(* CoDeSys 2.3.9.48 project: 5_hospital-Vyt_1Item.pro *)
(* Libraries: Standard.lib 8.11.10 13:37:48 *)

(* PLC configuration (modules and I/O channels)
_Y1_1 AT %QX0.0 [BOOLOnX_Q] Ch_1 Digital output
_Y2_1 AT %QX0.1 [BOOLOnX_Q] Ch_2 Digital output
_PCH1_1 AT %QX0.2 [BOOLOnX_Q] Ch_3 Digital output
_PCH2_1 AT %QX0.3 [BOOLOnX_Q] Ch_4 Digital output
AT %QX0.4 [BOOLOnX_Q] Ch_5 Digital output
AT %QX0.5 [BOOLOnX_Q] Ch_6 Digital output
AT %QX0.6 [BOOLOnX_Q] Ch_7 Digital output
AT %QX0.7 [BOOLOnX_Q] Ch_8 Digital output
_AlmN1_1 AT %IX0.0 [BOOLOnX_I] Ch_1 Digital input
_RotationInv1_1 AT %IX0.1 [BOOLOnX_I] Ch_2 Digital input
_AlmN2_1 AT %IX0.2 [BOOLOnX_I] Ch_3 Digital input
_RotationInv2_1 AT %IX0.3 [BOOLOnX_I] Ch_4 Digital input
_HeatProtectM1_1 AT %IX0.4 [BOOLOnX_I] Ch_5 Digital input
AT %IX0.5 [BOOLOnX_I] Ch_6 Digital input
_HeatProtectM2_1 AT %IX0.6 [BOOLOnX_I] Ch_7 Digital input
AT %IX0.7 [BOOLOnX_I] Ch_8 Digital input
Fieldbus variables [FB_VARS] node 1, in %IB0 out %QB0
Flag variables [FLAG_VARS] node 2, in %IB0 out %QB0
Modbus-Master [MB_MASTER] node 3, in %IB0 out %QB0
*)

(* Global variable list: _DO *)
VAR_GLOBAL
	Y1_1	:	BOOL;
	Y2_1	:	BOOL;

	PCH1_1	:	BOOL;
	PCH2_1	:	BOOL;


	Y1_2	:	BOOL;
	Y2_2	:	BOOL;

	PCH1_2	:	BOOL;
	PCH2_2	:	BOOL;


	Y1_3	:	BOOL;
	Y2_3	:	BOOL;

	PCH1_3	:	BOOL;
	PCH2_3	:	BOOL;

	Y1_4	:	BOOL;
	Y2_4	:	BOOL;

	PCH1_4	:	BOOL;
	PCH2_4	:	BOOL;

	wDO AT %MW1000: 	WORD;


END_VAR

(* Global variable list: Alm *)
VAR_GLOBAL

	xResetAllAlm AT %MW100: 	BOOL;
	xResetAlm_M1_1 AT %MW104:	BOOL;
	xResetAlm_M2_1 AT %MW108:	BOOL;

	wAlm_Motor_M1_1 AT %MW112: WORD;
	wAlm_Motor_M2_1 AT %MW116:	WORD;


	xResetAlm_M1_2 AT %MW120: BOOL;
	xResetAlm_M2_2 AT %MW124:	BOOL;

	wAlm_Motor_M1_2 AT %MW128: WORD;
	wAlm_Motor_M2_2 AT %MW132:	WORD;


	xResetAlm_M1_3 AT %MW136:	BOOL;
	xResetAlm_M2_3 AT %MW140:	BOOL;

	wAlm_Motor_M1_3 AT %MW144: WORD;
	wAlm_Motor_M2_3 AT %MW148:	WORD;

	xResetAlm_M1_4 AT %MW152:	BOOL;
	xResetAlm_M2_4 AT %MW156:	BOOL;

	wAlm_Motor_M1_4 AT %MW160: WORD;
	wAlm_Motor_M2_4 AT %MW164:	WORD;

END_VAR

(* Global variable list: DI *)
VAR_GLOBAL



	AlmN1_1	:	BOOL;
	AlmN2_1	:	BOOL;
	HeatProtectM1_1	:	BOOL;
	HeatProtectM2_1	:	BOOL;
	RotationInv1_1	:	BOOL;
	RotationInv2_1	:	BOOL;

	AlmN1_2	:	BOOL;
	AlmN2_2	:	BOOL;
	HeatProtectM1_2	:	BOOL;
	HeatProtectM2_2	:	BOOL;
	RotationInv1_2	:	BOOL;
	RotationInv2_2	:	BOOL;

	AlmN1_3	:	BOOL;
	AlmN2_3	:	BOOL;
	HeatProtectM1_3	:	BOOL;
	HeatProtectM2_3	:	BOOL;
	RotationInv1_3	:	BOOL;
	RotationInv2_3	:	BOOL;

	AlmN1_4	:	BOOL;
	AlmN2_4	:	BOOL;
	HeatProtectM1_4	:	BOOL;
	HeatProtectM2_4	:	BOOL;
	RotationInv1_4	:	BOOL;
	RotationInv2_4	:	BOOL;

	wDI_1 AT %MW1010: 	WORD;
	wDI_2 AT %MW1020: 	WORD;

END_VAR

(* Global variable list: Motors *)
VAR_GLOBAL
	xVentStart_1 AT %MW200:BOOL;
	xVentStart_2 AT %MW204:BOOL;
	xVentStart_3 AT %MW208:BOOL;
	xVentStart_4 AT %MW212:BOOL;
END_VAR

(* Global variable list: Settings *)
VAR_GLOBAL RETAIN

	xStartWithSecond_1 AT %MW300: BOOL;
	xStartWithSecond_2 AT %MW304: BOOL;
	xStartWithSecond_3 AT %MW308: BOOL;
	xStartWithSecond_4 AT %MW312: BOOL;

END_VAR

(* POU PLC_PRG, ST *)
PROGRAM PLC_PRG
VAR
	xFirstStart: BOOL:= TRUE;
END_VAR
InToVars();

IF xFirstStart THEN
	xFirstStart:=FALSE;
	xVentStart_1:=TRUE;
	xVentStart_2:=TRUE;
	xVentStart_3:=TRUE;
	xVentStart_4:=TRUE;
END_IF


prMotor_1();
(*
prMotor_2();
prMotor_3();
*)
xResetAllAlm:=FALSE;

VarsToOut();
END_PROGRAM

(* POU InToVars, ST *)
PROGRAM InToVars
VAR
END_VAR
AlmN1_1	:=	_AlmN1_1	;
AlmN2_1	:=	_AlmN2_1	;
HeatProtectM1_1	:=	_HeatProtectM1_1	;
HeatProtectM2_1	:=	_HeatProtectM2_1	;
RotationInv1_1	:=	_RotationInv1_1	;
RotationInv2_1	:=	_RotationInv2_1	;
(*
AlmN1_2	:=	_AlmN1_2	;
AlmN2_2	:=	_AlmN2_2	;
HeatProtectM1_2	:=	_HeatProtectM1_2	;
HeatProtectM2_2	:=	_HeatProtectM2_2	;
RotationInv1_2	:=	_RotationInv1_2	;
RotationInv2_2	:=	_RotationInv2_2	;
AlmN1_3	:=	_AlmN1_3	;
AlmN2_3	:=	_AlmN2_3	;
HeatProtectM1_3	:=	_HeatProtectM1_3	;
HeatProtectM2_3	:=	_HeatProtectM2_3	;
RotationInv1_3	:=	_RotationInv1_3	;
RotationInv2_3	:=	_RotationInv2_3	;
*)
(*
AlmN1_4	:=	_AlmN1_4	;
AlmN2_4	:=	_AlmN2_4	;
HeatProtectM1_4	:=	_HeatProtectM1_4	;
HeatProtectM2_4	:=	_HeatProtectM2_4	;
RotationInv1_4	:=	_RotationInv1_4	;
RotationInv2_4	:=	_RotationInv2_4;

*)
wDI_1.0	:=	AlmN1_1	;
wDI_1.1	:=	AlmN2_1	;
wDI_1.2	:=	HeatProtectM1_1	;
wDI_1.3	:=	HeatProtectM2_1	;
wDI_1.4	:=	RotationInv1_1	;
wDI_1.5	:=	RotationInv2_1	;
wDI_1.6	:=	AlmN1_2	;
wDI_1.7	:=	AlmN2_2	;
wDI_1.8	:=	HeatProtectM1_2	;
wDI_1.9	:=	HeatProtectM2_2	;
wDI_1.10	:=	RotationInv1_2	;
wDI_1.11	:=	RotationInv2_2	;
wDI_1.12	:=	AlmN1_3	;
wDI_1.13	:=	AlmN2_3	;
wDI_1.14	:=	HeatProtectM1_3	;
wDI_1.15	:=	HeatProtectM2_3	;
wDI_2.0	:=	RotationInv1_3	;
wDI_2.1	:=	RotationInv2_3	;
wDI_2.2	:=	AlmN1_4	;
wDI_2.3	:=	AlmN2_4	;
wDI_2.4	:=	HeatProtectM1_4	;
wDI_2.5	:=	HeatProtectM2_4	;
wDI_2.6	:=	RotationInv1_4	;
wDI_2.7	:=	RotationInv2_4	;
END_PROGRAM

(* POU Device/Motor/prMotor_1, ST *)
PROGRAM prMotor_1
VAR
	SwitchMotors: fbSwitchMotors;
	Motor1: fbMotor;
	Motor2: fbMotor;
	xStart_M1: BOOL;
	xStart_M2: BOOL;
END_VAR
SwitchMotors(
	xStartingMotorChoose:= xStartWithSecond_1,
	wAlmMotor_M1:= wAlm_Motor_M1_1,
	wAlmMotor_M2:= wAlm_Motor_M2_1,
	xStartVent:= xVentStart_1,
	xStartM1=>xStart_M1 ,
	xStartM2=> xStart_M2);

Motor1(
	Y1_isOn:=TRUE ,
	xFeadback:= AlmN1_1,
	HeatProtection:=(* HeatProtectM1_1*)TRUE,
	xInvAlm:=RotationInv1_1,
	xStart:= xStart_M1,
	xZaslOpn:= Y1_1,
	xResetAllAlm:= xResetAllAlm,
	xResetMyAlm:=xResetAlm_M1_1,
	MotorStart=> PCH1_1,
	wError=>wAlm_Motor_M1_1 );

Motor2(
	Y1_isOn:=TRUE ,
	xFeadback:= AlmN2_1,
	HeatProtection:= (*HeatProtectM2_1*)TRUE,
	xInvAlm:=RotationInv2_1,
	xStart:= xStart_M2,
	xZaslOpn:= Y2_1,
	xResetAllAlm:= xResetAllAlm,
	xResetMyAlm:=xResetAlm_M2_1,
	MotorStart=> PCH2_1,
	wError=>wAlm_Motor_M2_1 );
END_PROGRAM

(* POU Device/Motor/FB/fbSwitchMotors, ST *)
FUNCTION_BLOCK fbSwitchMotors
VAR_INPUT
	xStartingMotorChoose: BOOL;
	wAlmMotor_M1: WORD;
	wAlmMotor_M2: WORD;
	xStartVent:	BOOL;
END_VAR
VAR_OUTPUT
	xStartM1:	BOOL;
	xStartM2:	BOOL;
END_VAR
VAR
END_VAR
IF xStartVent THEN
	xStartM1:=((NOT xStartingMotorChoose) OR wAlmMotor_M2 > 0) AND  wAlmMotor_M1 = 0;
	xStartM2:=(xStartingMotorChoose OR wAlmMotor_M1 > 0) AND  wAlmMotor_M2 = 0;
ELSE
	xStartM1:=FALSE;
	xStartM2:=FALSE;
END_IF
END_FUNCTION_BLOCK

(* POU Device/Motor/FB/fbMotor, ST *)
FUNCTION_BLOCK fbMotor
VAR_INPUT
	Y1_isOn:	BOOL;
	xFeadback:	BOOL;
	xInvAlm:	BOOL;
	HeatProtection:	BOOL;

END_VAR
VAR_IN_OUT
	xStart: BOOL;
	xZaslOpn:	BOOL;
	xResetAllAlm:	BOOL;
	xResetMyAlm:	BOOL;
END_VAR
VAR_OUTPUT
	MotorStart:BOOL;
	wError:WORD;
END_VAR

VAR
	tnZaslOpn: TON;
	tnFeadbackAlm: TON;
END_VAR
wError.0:= NOT Y1_isOn;

wError.1:=NOT HeatProtection;

tnFeadbackAlm(IN:= MotorStart AND (NOT xFeadback), PT:=T#20s);
IF tnFeadbackAlm.Q THEN
	wError.2:=TRUE;
END_IF

IF xInvAlm THEN
	wError.4:=TRUE;
END_IF

xZaslOpn:= xStart AND wError =0;

tnZaslOpn(IN:=xZaslOpn, PT:=T#20S, Q=>MotorStart);

IF xResetAllAlm OR xResetMyAlm THEN
	wError:=0;
	xResetMyAlm:=FALSE;
END_IF
END_FUNCTION_BLOCK

(* POU VarsToOut, ST *)
PROGRAM VarsToOut
VAR
END_VAR
_Y1_1	:=	Y1_1	;
_Y2_1	:=	Y2_1	;
_PCH1_1	:=	PCH1_1	;
_PCH2_1	:=	PCH2_1	;
(*
_Y1_2	:=	Y1_2	;
_Y2_2	:=	Y2_2	;
_PCH1_2	:=	PCH1_2	;
_PCH2_2	:=	PCH2_2	;
_Y1_3	:=	Y1_3	;
_Y2_3	:=	Y2_3	;
_PCH1_3	:=	PCH1_3	;
_PCH2_3	:=	PCH2_3	;
*)
(*
_Y1_4	:=	Y1_4	;
_Y2_4	:=	Y2_4	;
_PCH1_4	:=	PCH1_4	;
_PCH2_4	:=	PCH2_4	;
*)
wDO.0	:=	Y1_1	;
wDO.1	:=	Y2_1	;
wDO.2	:=	PCH1_1	;
wDO.3	:=	PCH2_1	;
wDO.4	:=	Y1_2	;
wDO.5	:=	Y2_2	;
wDO.6	:=	PCH1_2	;
wDO.7	:=	PCH2_2	;
wDO.8	:=	Y1_3	;
wDO.9	:=	Y2_3	;
wDO.10	:=	PCH1_3	;
wDO.11	:=	PCH2_3	;
wDO.12	:=	Y1_4	;
wDO.13	:=	Y2_4	;
wDO.14	:=	PCH1_4	;
wDO.15	:=	PCH2_4	;
END_PROGRAM

(* POU Configuration/MODBUS_CONFIGURATION, ST *)
PROGRAM MODBUS_CONFIGURATION        
VAR                                
END_VAR                            
(*                                 
   <?xml version="1.0" encoding="UTF-16" standalone="yes"?>
<network xml_structure_version="1" xml_feature_version="1">
	<generator_settings minRTUTaskCycleTimeMs="5" minEthaskCycleTimeMs="5" ethSlaveMultiplier="0.1" rtuInterfaceMultiplier="0.1" taskGeneration="true"/>
</network>
                              
*)                                 
;                                  
END_PROGRAM

(* POU Device/Motor/prMotor_2, ST *)
PROGRAM prMotor_2
VAR
	SwitchMotors: fbSwitchMotors;
	Motor1: fbMotor;
	Motor2: fbMotor;
	xStart_M1: BOOL;
	xStart_M2: BOOL;
END_VAR
SwitchMotors(
	xStartingMotorChoose:= xStartWithSecond_2,
	wAlmMotor_M1:= wAlm_Motor_M1_2,
	wAlmMotor_M2:= wAlm_Motor_M2_2,
	xStartVent:= xVentStart_2,
	xStartM1=>xStart_M1 ,
	xStartM2=> xStart_M2);

Motor1(
	Y1_isOn:=TRUE ,
	xFeadback:= AlmN1_2,
	HeatProtection:= (*HeatProtectM1_2*)TRUE,
	xInvAlm:=RotationInv1_2,
	xStart:= xStart_M1,
	xZaslOpn:= Y1_2,
	xResetAllAlm:= xResetAllAlm,
	xResetMyAlm:=xResetAlm_M1_2,
	MotorStart=> PCH1_2,
	wError=>wAlm_Motor_M1_2 );

Motor2(
	Y1_isOn:=TRUE ,
	xFeadback:= AlmN2_2,
	HeatProtection:= (*HeatProtectM2_1*)TRUE,
	xInvAlm:=RotationInv2_2,
	xStart:= xStart_M2,
	xZaslOpn:= Y2_2,
	xResetAllAlm:= xResetAllAlm,
	xResetMyAlm:=xResetAlm_M2_2,
	MotorStart=> PCH2_2,
	wError=>wAlm_Motor_M2_2 );
END_PROGRAM

(* POU Device/Motor/prMotor_3, ST *)
PROGRAM prMotor_3
VAR
	SwitchMotors: fbSwitchMotors;
	Motor1: fbMotor;
	Motor2: fbMotor;
	xStart_M1: BOOL;
	xStart_M2: BOOL;
END_VAR
SwitchMotors(
	xStartingMotorChoose:= xStartWithSecond_3,
	wAlmMotor_M1:= wAlm_Motor_M1_3,
	wAlmMotor_M2:= wAlm_Motor_M2_3,
	xStartVent:= xVentStart_3,
	xStartM1=>xStart_M1 ,
	xStartM2=> xStart_M2);

Motor1(
	Y1_isOn:=TRUE ,
	xFeadback:= AlmN1_3,
	HeatProtection:=(* HeatProtectM1_3*)NOT RotationInv1_3,
	xInvAlm:=RotationInv1_3,
	xStart:= xStart_M1,
	xZaslOpn:= Y1_3,
	xResetAllAlm:= xResetAllAlm,
	xResetMyAlm:=xResetAlm_M1_3,
	MotorStart=> PCH1_3,
	wError=>wAlm_Motor_M1_3 );

Motor2(
	Y1_isOn:=TRUE ,
	xFeadback:= AlmN2_3,
	HeatProtection:= (*HeatProtectM2_1*)NOT RotationInv2_3,
	xStart:= xStart_M2,
	xZaslOpn:= Y2_3,
	xResetAllAlm:= xResetAllAlm,
	xResetMyAlm:=xResetAlm_M2_3,
	MotorStart=> PCH2_3,
	wError=>wAlm_Motor_M2_3 );
END_PROGRAM
